KUKA KRL data list: ps_com_geo_c1.dat

&ACCESS RVO1
&REL 24
&COMMENT Solda GUN C1 Geometria
&PARAM DISKPATH = KRC:\R1\Program\SOLDA LTC
DEFDAT  ps_com_geo_c1
;FOLD EXTERNAL DECLARATIONS;%{PE}%MKUKATPBASIS,%CEXT,%VCOMMON,%P
;FOLD GRIPPERTECH EXT
EXT  H50 (INT  :IN,INT  :IN,INT  :IN,GRP_TYP  :IN )
;ENDFOLD (GRIPPERTECH EXT)
;FOLD SPOTTECH EXT
EXT  USERSPOT (S_COMMAND  :IN,SPOT_TYPE  :IN )
;ENDFOLD (SPOTTECH EXT)
;FOLD BASISTECH EXT;%{PE}%MKUKATPBASIS,%CEXT,%VEXT,%P
EXT  BAS (BAS_COMMAND  :IN,REAL  :IN )
DECL INT SUCCESS
;ENDFOLD (BASISTECH EXT)
;FOLD USER EXT;%{E}%MKUKATPUSER,%CEXT,%VEXT,%P
;Make your modifications here

;ENDFOLD (USER EXT)
;ENDFOLD (EXTERNAL DECLARATIONS)

;# ============ START PATH : swp_p13050r4_com_geo_c1 =============
DECL FDAT Fs_lx488={TOOL_NO 1,BASE_NO 1,IPO_FRAME #BASE,POINT2[] " "}
DECL PDAT PP_OLP5={VEL 100.0,ACC 100.0,APO_DIST 100.0,APO_MODE #CDIS}
DECL E6POS Xs_lx488={X -360.817993,Y 965.559021,Z 683.950989,A 93.2594986,B 64.8991013,C -75.3226013,S 2,T 10,E1 4060.29907,E2 0.0,E3 0.0,E4 0.0,E5 0.0,E6 0.0}
DECL FDAT Fswp_60_5140={TOOL_NO 1,BASE_NO 1,IPO_FRAME #BASE,POINT2[] " "}
DECL PDAT PP_OLP7={VEL 100.0,ACC 100.0,APO_DIST 0.0}
DECL SPOT_TYPE SS_OLP1={GUN 1,PAIR #FIRST,RETR #CLO,CLO_TM 0,PGNO1 1,PRESS1 1.0,PGNO2 0,PRESS2 0.0}
DECL E6POS Xswp_60_5140={X 136.687195,Y 902.795288,Z 579.572021,A 83.2147293,B 65.6525803,C -84.4438324,S 2,T 10,E1 4060.30103,E2 0.0,E3 0.0,E4 0.0,E5 0.0,E6 0.0}
DECL FDAT Fs_lx486={TOOL_NO 1,BASE_NO 1,IPO_FRAME #BASE,POINT2[] " "}
DECL PDAT PP_OLP9={VEL 100.0,ACC 100.0,APO_DIST 100.0,APO_MODE #CDIS}
DECL E6POS Xs_lx486={X -360.820007,Y 965.559998,Z 683.950989,A 93.2594986,B 64.8992004,C -75.3226013,S 2,T 10,E1 4060.29907,E2 0.0,E3 0.0,E4 0.0,E5 0.0,E6 0.0}
DECL PDAT PP_OLP10={VEL 100.0,ACC 100.0,APO_DIST 50.0,APO_MODE #CDIS}
DECL FDAT Fswp_60_5118={TOOL_NO 1,BASE_NO 1,IPO_FRAME #BASE,POINT2[] " "}
DECL PDAT PP_OLP12={VEL 100.0,ACC 100.0,APO_DIST 0.0}
DECL SPOT_TYPE SS_OLP2={GUN 1,PAIR #FIRST,RETR #CLO,CLO_TM 0,PGNO1 1,PRESS1 1.0,PGNO2 0,PRESS2 0.0}
DECL E6POS Xswp_60_5118={X 94.381012,Y 322.608704,Z 577.968018,A 0.639736116,B 88.9835663,C -175.218796,S 2,T 10,E1 4060.29199,E2 0.0,E3 0.0,E4 0.0,E5 0.0,E6 0.0}
DECL PDAT PP_OLP14={VEL 100.0,ACC 100.0,APO_DIST 100.0,APO_MODE #CDIS}
DECL PDAT PP_OLP16={VEL 100.0,ACC 100.0,APO_DIST 100.0,APO_MODE #CDIS}
DECL FDAT Fswp_60_5026={TOOL_NO 1,BASE_NO 1,IPO_FRAME #BASE,POINT2[] " "}
DECL PDAT PP_OLP18={VEL 100.0,ACC 100.0,APO_DIST 0.0}
DECL SPOT_TYPE SS_OLP3={GUN 1,PAIR #FIRST,RETR #CLO,CLO_TM 0,PGNO1 1,PRESS1 1.0,PGNO2 0,PRESS2 0.0}
DECL E6POS Xswp_60_5026={X 159.332901,Y 427.524109,Z 4.32035685,A 90.0029831,B -50.8949509,C -90.0011292,S 2,T 42,E1 4060.2771,E2 0.0,E3 0.0,E4 0.0,E5 0.0,E6 0.0}
DECL FDAT Fswp_60_5020={TOOL_NO 1,BASE_NO 1,IPO_FRAME #BASE,POINT2[] " "}
DECL PDAT PP_OLP19={VEL 100.0,ACC 100.0,APO_DIST 0.0}
DECL SPOT_TYPE SS_OLP4={GUN 1,PAIR #FIRST,RETR #CLO,CLO_TM 0,PGNO1 1,PRESS1 1.0,PGNO2 0,PRESS2 0.0}
DECL E6POS Xswp_60_5020={X 158.871796,Y 329.765594,Z 2.61356592,A 90.0077286,B -48.4540215,C -90.0015869,S 2,T 42,E1 4060.2981,E2 0.0,E3 0.0,E4 0.0,E5 0.0,E6 0.0}
DECL FDAT Fswp_60_5016={TOOL_NO 1,BASE_NO 1,IPO_FRAME #BASE,POINT2[] " "}
DECL PDAT PP_OLP20={VEL 100.0,ACC 100.0,APO_DIST 0.0}
DECL SPOT_TYPE SS_OLP5={GUN 1,PAIR #FIRST,RETR #CLO,CLO_TM 0,PGNO1 1,PRESS1 1.0,PGNO2 0,PRESS2 0.0}
DECL E6POS Xswp_60_5016={X 159.657196,Y 262.3927,Z 3.53638506,A 90.0078125,B -48.4543304,C -90.0026169,S 2,T 42,E1 4060.2959,E2 0.0,E3 0.0,E4 0.0,E5 0.0,E6 0.0}
DECL FDAT Fswp_60_5014={TOOL_NO 1,BASE_NO 1,IPO_FRAME #BASE,POINT2[] " "}
DECL PDAT PP_OLP21={VEL 100.0,ACC 100.0,APO_DIST 0.0}
DECL SPOT_TYPE SS_OLP6={GUN 1,PAIR #FIRST,RETR #CLO,CLO_TM 0,PGNO1 1,PRESS1 1.0,PGNO2 0,PRESS2 0.0}
DECL E6POS Xswp_60_5014={X 159.661102,Y 231.6185,Z 3.63049507,A 90.0080414,B -48.4544716,C -90.0028687,S 2,T 42,E1 4060.29712,E2 0.0,E3 0.0,E4 0.0,E5 0.0,E6 0.0}
DECL PDAT PP_OLP22={VEL 100.0,ACC 100.0,APO_DIST 100.0,APO_MODE #CDIS}
DECL FDAT Fs_lx470={TOOL_NO 1,BASE_NO 1,IPO_FRAME #BASE,POINT2[] " "}
DECL PDAT PP_OLP23={VEL 100.0,ACC 100.0,APO_DIST 100.0,APO_MODE #CDIS}
DECL E6POS Xs_lx470={X -243.503998,Y 293.677002,Z -34.257,A 90.0,B -44.5937996,C -90.0,S 2,T 10,E1 4060.29907,E2 0.0,E3 0.0,E4 0.0,E5 0.0,E6 0.0}
DECL PDAT PP_OLP24={VEL 100.0,ACC 100.0,APO_DIST 100.0,APO_MODE #CDIS}
DECL FDAT Flx507={TOOL_NO 1,BASE_NO 1,IPO_FRAME #BASE,POINT2[] " "}
DECL PDAT PP_OLP25={VEL 100.0,ACC 100.0,APO_DIST 100.0,APO_MODE #CDIS}
DECL E6POS Xlx507={X -11.6990004,Y 1057.32996,Z -233.384003,A 68.1399002,B -45.7775993,C -90.0,S 2,T 10,E1 4060.29907,E2 0.0,E3 0.0,E4 0.0,E5 0.0,E6 0.0}
DECL PDAT PP_OLP26={VEL 100.0,ACC 100.0,APO_DIST 100.0,APO_MODE #CDIS}
DECL FDAT Fswp_60_5042={TOOL_NO 1,BASE_NO 1,IPO_FRAME #BASE,POINT2[] " "}
DECL PDAT PP_OLP27={VEL 100.0,ACC 100.0,APO_DIST 0.0}
DECL SPOT_TYPE SS_OLP7={GUN 1,PAIR #FIRST,RETR #CLO,CLO_TM 0,PGNO1 1,PRESS1 1.0,PGNO2 0,PRESS2 0.0}
DECL E6POS Xswp_60_5042={X 176.981293,Y 1036.93799,Z -181.563095,A 68.1404114,B -45.7783699,C -90.0011597,S 2,T 10,E1 4060.30005,E2 0.0,E3 0.0,E4 0.0,E5 0.0,E6 0.0}
DECL FDAT Fswp_60_5040={TOOL_NO 1,BASE_NO 1,IPO_FRAME #BASE,POINT2[] " "}
DECL PDAT PP_OLP28={VEL 100.0,ACC 100.0,APO_DIST 0.0}
DECL SPOT_TYPE SS_OLP8={GUN 1,PAIR #FIRST,RETR #CLO,CLO_TM 0,PGNO1 1,PRESS1 1.0,PGNO2 0,PRESS2 0.0}
DECL E6POS Xswp_60_5040={X 172.178604,Y 1008.79102,Z -183.401794,A 176.628098,B -88.2014084,C 167.694305,S 2,T 10,E1 4060.30103,E2 0.0,E3 0.0,E4 0.0,E5 0.0,E6 0.0}
DECL FDAT Fswp_60_5038={TOOL_NO 1,BASE_NO 1,IPO_FRAME #BASE,POINT2[] " "}
DECL PDAT PP_OLP29={VEL 100.0,ACC 100.0,APO_DIST 0.0}
DECL SPOT_TYPE SS_OLP9={GUN 1,PAIR #FIRST,RETR #CLO,CLO_TM 0,PGNO1 1,PRESS1 1.0,PGNO2 0,PRESS2 0.0}
DECL E6POS Xswp_60_5038={X 164.622696,Y 982.143127,Z -183.500595,A -120.116699,B -89.1609726,C 109.444,S 2,T 10,E1 4060.29907,E2 0.0,E3 0.0,E4 0.0,E5 0.0,E6 0.0}
DECL FDAT Fswp_60_5036={TOOL_NO 1,BASE_NO 1,IPO_FRAME #BASE,POINT2[] " "}
DECL SPOT_TYPE SS_OLP10={GUN 1,PAIR #FIRST,RETR #CLO,CLO_TM 0,PGNO1 1,PRESS1 1.0,PGNO2 0,PRESS2 0.0}
DECL E6POS Xswp_60_5036={X 179.731094,Y 901.85553,Z -137.682495,A -105.0299,B -89.9987488,C 105.028702,S 2,T 42,E1 4060.29907,E2 0.0,E3 0.0,E4 0.0,E5 0.0,E6 0.0}
DECL FDAT Fswp_60_5028={TOOL_NO 1,BASE_NO 1,IPO_FRAME #BASE,POINT2[] " "}
DECL PDAT PP_OLP32={VEL 100.0,ACC 100.0,APO_DIST 0.0}
DECL SPOT_TYPE SS_OLP11={GUN 1,PAIR #FIRST,RETR #CLO,CLO_TM 0,PGNO1 1,PRESS1 1.0,PGNO2 0,PRESS2 0.0}
DECL E6POS Xswp_60_5028={X 182.583893,Y 794.820129,Z -47.8096008,A -163.747406,B -89.5717773,C 163.750702,S 2,T 42,E1 4060.29395,E2 0.0,E3 0.0,E4 0.0,E5 0.0,E6 0.0}
DECL FDAT Fs_lx464={TOOL_NO 1,BASE_NO 1,IPO_FRAME #BASE,POINT2[] " "}
DECL PDAT PP_OLP33={VEL 100.0,ACC 100.0,APO_DIST 100.0,APO_MODE #CDIS}
DECL E6POS Xs_lx464={X 178.498993,Y 805.025024,Z -118.82,A 0.0,B -90.0,C 0.0,S 2,T 42,E1 4060.29907,E2 0.0,E3 0.0,E4 0.0,E5 0.0,E6 0.0}
DECL PDAT PP_OLP34={VEL 100.0,ACC 100.0,APO_DIST 100.0,APO_MODE #CDIS}
DECL SPOT_TYPE SS_OLP12={GUN 1,PAIR #FIRST,RETR #CLO,CLO_TM 0,PGNO1 1,PRESS1 1.0,PGNO2 0,PRESS2 0.0}
DECL FDAT Fswp_60_5203={TOOL_NO 1,BASE_NO 1,IPO_FRAME #BASE,POINT2[] " "}
DECL SPOT_TYPE SS_OLP13={GUN 1,PAIR #FIRST,RETR #CLO,CLO_TM 0,PGNO1 1,PRESS1 1.0,PGNO2 0,PRESS2 0.0}
DECL E6POS Xswp_60_5203={X 156.1819,Y 485.568604,Z 388.023712,A 90.0274734,B -54.6427803,C -86.9009323,S 2,T 10,E1 4060.31592,E2 0.0,E3 0.0,E4 0.0,E5 0.0,E6 0.0}
DECL FDAT Fswp_60_5195={TOOL_NO 1,BASE_NO 1,IPO_FRAME #BASE,POINT2[] " "}
DECL SPOT_TYPE SS_OLP14={GUN 1,PAIR #FIRST,RETR #CLO,CLO_TM 0,PGNO1 1,PRESS1 1.0,PGNO2 0,PRESS2 0.0}
DECL E6POS Xswp_60_5195={X 161.142303,Y 202.515198,Z 386.019104,A -88.2071686,B -36.5904808,C 88.8797302,S 2,T 10,E1 4060.31396,E2 0.0,E3 0.0,E4 0.0,E5 0.0,E6 0.0}
DECL FDAT Fswp_60_5190={TOOL_NO 1,BASE_NO 1,IPO_FRAME #BASE,POINT2[] " "}
DECL SPOT_TYPE SS_OLP15={GUN 1,PAIR #FIRST,RETR #CLO,CLO_TM 0,PGNO1 1,PRESS1 1.0,PGNO2 0,PRESS2 0.0}
DECL E6POS Xswp_60_5190={X 161.480301,Y 148.9478,Z 280.717194,A -89.3926468,B -1.94816995,C 88.6738968,S 2,T 10,E1 4060.31494,E2 0.0,E3 0.0,E4 0.0,E5 0.0,E6 0.0}
DECL FDAT Fswp_60_5218={TOOL_NO 1,BASE_NO 1,IPO_FRAME #BASE,POINT2[] " "}
DECL SPOT_TYPE SS_OLP16={GUN 1,PAIR #FIRST,RETR #CLO,CLO_TM 0,PGNO1 1,PRESS1 1.0,PGNO2 0,PRESS2 0.0}
DECL E6POS Xswp_60_5218={X 164.738403,Y 122.212402,Z 106.1138,A -90.9965591,B 31.5576591,C 87.71698,S 2,T 10,E1 4060.31396,E2 0.0,E3 0.0,E4 0.0,E5 0.0,E6 0.0}
DECL PDAT PP_OLP52={VEL 100.0,ACC 100.0,APO_DIST 100.0,APO_MODE #CDIS}
DECL SPOT_TYPE SS_OLP17={GUN 1,PAIR #FIRST,RETR #CLO,CLO_TM 0,PGNO1 1,PRESS1 1.0,PGNO2 0,PRESS2 0.0}
DECL SPOT_TYPE SS_OLP18={GUN 1,PAIR #FIRST,RETR #CLO,CLO_TM 0,PGNO1 1,PRESS1 1.0,PGNO2 0,PRESS2 0.0}
DECL SPOT_TYPE SS_OLP19={GUN 1,PAIR #FIRST,RETR #CLO,CLO_TM 0,PGNO1 1,PRESS1 1.0,PGNO2 0,PRESS2 0.0}
DECL FDAT Fswp_60_5066={TOOL_NO 1,BASE_NO 1,IPO_FRAME #BASE,POINT2[] " "}
DECL SPOT_TYPE SS_OLP20={GUN 1,PAIR #FIRST,RETR #CLO,CLO_TM 0,PGNO1 1,PRESS1 1.0,PGNO2 0,PRESS2 0.0}
DECL E6POS Xswp_60_5066={X 151.353302,Y 626.425415,Z 250.5159,A -92.1195831,B 18.5633907,C 91.8053436,S 2,T 10,E1 4060.30591,E2 0.0,E3 0.0,E4 0.0,E5 0.0,E6 0.0}
DECL PDAT PP_OLP59={VEL 100.0,ACC 100.0,APO_DIST 20.0,APO_MODE #CDIS}
DECL PDAT PP_OLP60={VEL 100.0,ACC 100.0,APO_DIST 20.0,APO_MODE #CDIS}
DECL PDAT PP_OLP61={VEL 100.0,ACC 100.0,APO_DIST 20.0,APO_MODE #CDIS}
DECL FDAT Fswp_60_5076={TOOL_NO 1,BASE_NO 1,IPO_FRAME #BASE,POINT2[] " "}
DECL PDAT PP_OLP63={VEL 100.0,ACC 100.0,APO_DIST 0.0}
DECL SPOT_TYPE SS_OLP21={GUN 1,PAIR #FIRST,RETR #CLO,CLO_TM 0,PGNO1 1,PRESS1 1.0,PGNO2 0,PRESS2 0.0}
DECL E6POS Xswp_60_5076={X 154.796707,Y 782.258972,Z 101.740097,A 87.1909637,B 70.1359329,C -93.0589066,S 2,T 10,E1 4060.29199,E2 0.0,E3 0.0,E4 0.0,E5 0.0,E6 0.0}
DECL PDAT PP_OLP64={VEL 100.0,ACC 100.0,APO_DIST 100.0,APO_MODE #CDIS}
DECL SPOT_TYPE SS_OLP22={GUN 1,PAIR #FIRST,RETR #CLO,CLO_TM 0,PGNO1 1,PRESS1 1.0,PGNO2 0,PRESS2 0.0}
DECL PDAT PP_OLP69={VEL 100.0,ACC 100.0,APO_DIST 100.0,APO_MODE #CDIS}
DECL PDAT PP_OLP72={VEL 100.0,ACC 100.0,APO_DIST 100.0,APO_MODE #CDIS}
DECL FDAT Fswp_60_5626={TOOL_NO 1,BASE_NO 1,IPO_FRAME #BASE,POINT2[] " "}
DECL PDAT PP_OLP73={VEL 100.0,ACC 100.0,APO_DIST 0.0}
DECL SPOT_TYPE SS_OLP23={GUN 1,PAIR #FIRST,RETR #CLO,CLO_TM 0,PGNO1 1,PRESS1 1.0,PGNO2 0,PRESS2 0.0}
DECL E6POS Xswp_60_5626={X 634.33252,Y 1098.11096,Z 1372.00806,A -179.633102,B -69.9991837,C 90.5753021,S 2,T 2,E1 5254.49902,E2 0.0,E3 0.0,E4 0.0,E5 0.0,E6 0.0}
DECL FDAT Fswp_60_5640={TOOL_NO 1,BASE_NO 1,IPO_FRAME #BASE,POINT2[] " "}
DECL PDAT PP_OLP74={VEL 100.0,ACC 100.0,APO_DIST 0.0}
DECL SPOT_TYPE SS_OLP24={GUN 1,PAIR #FIRST,RETR #CLO,CLO_TM 0,PGNO1 1,PRESS1 1.0,PGNO2 0,PRESS2 0.0}
DECL E6POS Xswp_60_5640={X 731.3703,Y 1097.53699,Z 1377.57104,A 0.929155171,B -80.0200806,C -89.9900208,S 2,T 2,E1 5254.5,E2 0.0,E3 0.0,E4 0.0,E5 0.0,E6 0.0}
DECL PDAT PP_OLP75={VEL 100.0,ACC 100.0,APO_DIST 100.0,APO_MODE #CDIS}
DECL PDAT PP_OLP76={VEL 100.0,ACC 100.0,APO_DIST 100.0,APO_MODE #CDIS}
DECL PDAT PP_OLP77={VEL 100.0,ACC 100.0,APO_DIST 50.0,APO_MODE #CDIS}
DECL PDAT PP_OLP78={VEL 100.0,ACC 100.0,APO_DIST 50.0,APO_MODE #CDIS}
DECL FDAT Fswp_60_5060={TOOL_NO 1,BASE_NO 1,IPO_FRAME #BASE,POINT2[] " "}
DECL PDAT PP_OLP79={VEL 100.0,ACC 100.0,APO_DIST 0.0}
DECL SPOT_TYPE SS_OLP25={GUN 1,PAIR #FIRST,RETR #CLO,CLO_TM 0,PGNO1 1,PRESS1 1.0,PGNO2 0,PRESS2 0.0}
DECL E6POS Xswp_60_5060={X 440.014313,Y 1093.56006,Z -44.92976,A -177.803696,B 33.6436501,C 90.0005798,S 2,T 34,E1 5251.46289,E2 0.0,E3 0.0,E4 0.0,E5 0.0,E6 0.0}
DECL PDAT PP_OLP80={VEL 100.0,ACC 100.0,APO_DIST 50.0,APO_MODE #CDIS}
DECL PDAT PP_OLP81={VEL 100.0,ACC 100.0,APO_DIST 50.0,APO_MODE #CDIS}
DECL PDAT PP_OLP82={VEL 100.0,ACC 100.0,APO_DIST 100.0,APO_MODE #CDIS}
DECL FDAT Fswp_60_5056={TOOL_NO 1,BASE_NO 1,IPO_FRAME #BASE,POINT2[] " "}
DECL PDAT PP_OLP85={VEL 100.0,ACC 100.0,APO_DIST 0.0}
DECL SPOT_TYPE SS_OLP26={GUN 1,PAIR #FIRST,RETR #CLO,CLO_TM 0,PGNO1 1,PRESS1 1.0,PGNO2 0,PRESS2 0.0}
DECL E6POS Xswp_60_5056={X 372.068909,Y 1092.44397,Z -181.150497,A 178.998093,B -2.52557802,C 89.9496765,S 2,T 34,E1 5252.67188,E2 0.0,E3 0.0,E4 0.0,E5 0.0,E6 0.0}
DECL FDAT Fswp_60_5058={TOOL_NO 1,BASE_NO 1,IPO_FRAME #BASE,POINT2[] " "}
DECL PDAT PP_OLP86={VEL 100.0,ACC 100.0,APO_DIST 0.0}
DECL SPOT_TYPE SS_OLP27={GUN 1,PAIR #FIRST,RETR #CLO,CLO_TM 0,PGNO1 1,PRESS1 1.0,PGNO2 0,PRESS2 0.0}
DECL E6POS Xswp_60_5058={X 404.384796,Y 1091.41699,Z -160.593002,A 178.922501,B -10.25455,C 90.7412491,S 2,T 34,E1 5253.80078,E2 0.0,E3 0.0,E4 0.0,E5 0.0,E6 0.0}
DECL PDAT PP_OLP88={VEL 100.0,ACC 100.0,APO_DIST 100.0,APO_MODE #CDIS}
DECL PDAT PP_OLP89={VEL 100.0,ACC 100.0,APO_DIST 100.0,APO_MODE #CDIS}
DECL FDAT Fswp_60_5424={TOOL_NO 1,BASE_NO 1,IPO_FRAME #BASE,POINT2[] " "}
DECL PDAT PP_OLP91={VEL 100.0,ACC 100.0,APO_DIST 0.0}
DECL SPOT_TYPE SS_OLP28={GUN 1,PAIR #FIRST,RETR #CLO,CLO_TM 0,PGNO1 1,PRESS1 1.0,PGNO2 0,PRESS2 0.0}
DECL E6POS Xswp_60_5424={X 1302.37805,Y 1186.15405,Z -56.5237999,A -0.546349108,B -50.1205597,C -90.0004196,S 2,T 2,E1 5251.78613,E2 0.0,E3 0.0,E4 0.0,E5 0.0,E6 0.0}
DECL PDAT PP_OLP92={VEL 100.0,ACC 100.0,APO_DIST 100.0,APO_MODE #CDIS}
DECL PDAT PP_OLP93={VEL 100.0,ACC 100.0,APO_DIST 100.0,APO_MODE #CDIS}
DECL PDAT PP_OLP96={VEL 100.0,ACC 100.0,APO_DIST 100.0,APO_MODE #CDIS}
DECL PDAT PP_OLP97={VEL 100.0,ACC 100.0,APO_DIST 20.0,APO_MODE #CDIS}
DECL FDAT Fswp_60_5430={TOOL_NO 1,BASE_NO 1,IPO_FRAME #BASE,POINT2[] " "}
DECL PDAT PP_OLP100={VEL 100.0,ACC 100.0,APO_DIST 0.0}
DECL SPOT_TYPE SS_OLP29={GUN 1,PAIR #FIRST,RETR #CLO,CLO_TM 0,PGNO1 1,PRESS1 1.0,PGNO2 0,PRESS2 0.0}
DECL E6POS Xswp_60_5430={X 1286.38098,Y 1123.69702,Z 5.72508383,A -0.644820571,B 48.2571411,C -90.0793915,S 2,T 2,E1 6178.22119,E2 0.0,E3 0.0,E4 0.0,E5 0.0,E6 0.0}
DECL FDAT Fswp_60_5432={TOOL_NO 1,BASE_NO 1,IPO_FRAME #BASE,POINT2[] " "}
DECL PDAT PP_OLP101={VEL 100.0,ACC 100.0,APO_DIST 0.0}
DECL SPOT_TYPE SS_OLP30={GUN 1,PAIR #FIRST,RETR #CLO,CLO_TM 0,PGNO1 1,PRESS1 1.0,PGNO2 0,PRESS2 0.0}
DECL E6POS Xswp_60_5432={X 1304.38,Y 1123.71106,Z 21.1026192,A -0.644798875,B 48.25737,C -90.0797424,S 2,T 2,E1 6217.10498,E2 0.0,E3 0.0,E4 0.0,E5 0.0,E6 0.0}
DECL FDAT Fswp_60_5434={TOOL_NO 1,BASE_NO 1,IPO_FRAME #BASE,POINT2[] " "}
DECL PDAT PP_OLP102={VEL 100.0,ACC 100.0,APO_DIST 0.0}
DECL SPOT_TYPE SS_OLP31={GUN 1,PAIR #FIRST,RETR #CLO,CLO_TM 0,PGNO1 1,PRESS1 1.0,PGNO2 0,PRESS2 0.0}
DECL E6POS Xswp_60_5434={X 1288.31995,Y 1122.44202,Z 30.7160091,A -0.641988695,B 48.2577095,C -90.0761871,S 2,T 2,E1 6172.71387,E2 0.0,E3 0.0,E4 0.0,E5 0.0,E6 0.0}
DECL FDAT Fswp_60_5436={TOOL_NO 1,BASE_NO 1,IPO_FRAME #BASE,POINT2[] " "}
DECL PDAT PP_OLP105={VEL 100.0,ACC 100.0,APO_DIST 0.0}
DECL SPOT_TYPE SS_OLP32={GUN 1,PAIR #FIRST,RETR #CLO,CLO_TM 0,PGNO1 1,PRESS1 1.0,PGNO2 0,PRESS2 0.0}
DECL E6POS Xswp_60_5436={X 1304.93005,Y 1120.12903,Z 80.8903885,A -0.630691886,B 29.8777504,C -90.0939484,S 2,T 2,E1 6169.68115,E2 0.0,E3 0.0,E4 0.0,E5 0.0,E6 0.0}
DECL FDAT Fswp_60_5438={TOOL_NO 1,BASE_NO 1,IPO_FRAME #BASE,POINT2[] " "}
DECL PDAT PP_OLP107={VEL 100.0,ACC 100.0,APO_DIST 0.0}
DECL SPOT_TYPE SS_OLP33={GUN 1,PAIR #FIRST,RETR #CLO,CLO_TM 0,PGNO1 1,PRESS1 1.0,PGNO2 0,PRESS2 0.0}
DECL E6POS Xswp_60_5438={X 1335.14502,Y 1125.09802,Z 99.5109024,A -0.583152175,B 19.4271107,C -90.0527191,S 2,T 2,E1 5977.15283,E2 0.0,E3 0.0,E4 0.0,E5 0.0,E6 0.0}
DECL FDAT Fswp_60_5440={TOOL_NO 1,BASE_NO 1,IPO_FRAME #BASE,POINT2[] " "}
DECL PDAT PP_OLP108={VEL 100.0,ACC 100.0,APO_DIST 0.0}
DECL SPOT_TYPE SS_OLP34={GUN 1,PAIR #FIRST,RETR #CLO,CLO_TM 0,PGNO1 1,PRESS1 1.0,PGNO2 0,PRESS2 0.0}
DECL E6POS Xswp_60_5440={X 1334.10596,Y 1122.04004,Z 140.932205,A -0.565891325,B -2.25514102,C -90.0501328,S 2,T 2,E1 5826.48584,E2 0.0,E3 0.0,E4 0.0,E5 0.0,E6 0.0}
DECL PDAT PP_OLP109={VEL 100.0,ACC 100.0,APO_DIST 100.0,APO_MODE #CDIS}
DECL PDAT PP_OLP110={VEL 100.0,ACC 100.0,APO_DIST 100.0,APO_MODE #CDIS}
DECL PDAT PP_OLP111={VEL 100.0,ACC 100.0,APO_DIST 100.0,APO_MODE #CDIS}
DECL PDAT PP_OLP112={VEL 100.0,ACC 100.0,APO_DIST 100.0,APO_MODE #CDIS}
DECL PDAT PP_OLP113={VEL 100.0,ACC 100.0,APO_DIST 0.0,APO_MODE #CDIS}
DECL BASIS_SUGG_T LAST_BASIS={POINT1[] "P0                      ",POINT2[] "P0                      ",CP_PARAMS[] "CPDAT0                  ",PTP_PARAMS[] "PDAT0                   ",CONT[] "                        ",CP_VEL[] "2.0                     ",PTP_VEL[] " 100                    ",SYNC_PARAMS[] "SYNCDAT                 ",SPL_NAME[] "S0                      "}
DECL FDAT FXs_lx487={TOOL_NO 1,BASE_NO 1,IPO_FRAME #BASE,POINT2[] " ",TQ_STATE FALSE}
DECL E6POS XXS_LX487={X 142.0215,Y 865.563782,Z 629.299988,A 92.7790527,B 65.0505371,C -75.8403931,S 2,T 10,E1 4060.29395,E2 0.0,E3 0.0,E4 0.0,E5 0.0,E6 0.0}
DECL PDAT PPDAT2={VEL 100.0,ACC 100.0,APO_DIST 100.0,APO_MODE #CDIS}
DECL E6POS XXS_LX502={X 142.021301,Y 865.560791,Z 629.294983,A 92.7791138,B 65.0502167,C -75.8401871,S 2,T 10,E1 4060.29395,E2 0.0,E3 0.0,E4 0.0,E5 0.0,E6 0.0}
DECL FDAT FXs_lx502={TOOL_NO 1,BASE_NO 1,IPO_FRAME #BASE,POINT2[] " ",TQ_STATE FALSE}
DECL PDAT PPDAT6={VEL 100.0,ACC 100.0,APO_DIST 100.0,APO_MODE #CDIS}
DECL E6POS XXS_LX484={X -406.284088,Y 364.974487,Z 582.284119,A -59.6039505,B 89.6699677,C 128.917496,S 2,T 10,E1 4060.2981,E2 0.0,E3 0.0,E4 0.0,E5 0.0,E6 0.0}
DECL FDAT FXs_lx484={TOOL_NO 1,BASE_NO 1,IPO_FRAME #BASE,POINT2[] " ",TQ_STATE FALSE}
DECL E6POS XXS_LX504={X 102.534103,Y 321.186096,Z 604.033508,A 152.166595,B 89.932457,C -19.8392105,S 2,T 10,E1 4060.30005,E2 0.0,E3 0.0,E4 0.0,E5 0.0,E6 0.0}
DECL FDAT FXs_lx504={TOOL_NO 1,BASE_NO 1,IPO_FRAME #BASE,POINT2[] " ",TQ_STATE FALSE}
DECL PDAT PPDAT8={VEL 100.0,ACC 100.0,APO_DIST 50.0,APO_MODE #CDIS}
DECL E6POS XXS_LX506={X 101.603203,Y 324.702209,Z 606.954773,A -105.589798,B 89.533989,C 82.46315,S 2,T 10,E1 4060.29907,E2 0.0,E3 0.0,E4 0.0,E5 0.0,E6 0.0}
DECL FDAT FXs_lx506={TOOL_NO 1,BASE_NO 1,IPO_FRAME #BASE,POINT2[] " ",TQ_STATE FALSE}
DECL PDAT PPDAT10={VEL 100.0,ACC 100.0,APO_DIST 100.0,APO_MODE #CDIS}
DECL E6POS XXS_LX482={X -401.920288,Y 344.626587,Z 598.098022,A -123.613403,B 89.7013168,C 73.3319473,S 2,T 10,E1 4060.2981,E2 0.0,E3 0.0,E4 0.0,E5 0.0,E6 0.0}
DECL FDAT FXs_lx482={TOOL_NO 1,BASE_NO 1,IPO_FRAME #BASE,POINT2[] " ",TQ_STATE FALSE}
DECL E6POS XXS_LX510={X 164.903503,Y 407.34549,Z -24.669241,A 90.0030136,B -50.8949699,C -90.0012512,S 2,T 42,E1 4060.2771,E2 0.0,E3 0.0,E4 0.0,E5 0.0,E6 0.0}
DECL FDAT FXs_lx510={TOOL_NO 1,BASE_NO 1,IPO_FRAME #BASE,POINT2[] " ",TQ_STATE FALSE}
DECL PDAT PPDAT14={VEL 100.0,ACC 100.0,APO_DIST 100.0,APO_MODE #CDIS}
DECL E6POS XXS_LX469={X 176.571396,Y 282.161896,Z -22.7473507,A 89.9942474,B -44.593441,C -89.9960175,S 2,T 42,E1 4060.30103,E2 0.0,E3 0.0,E4 0.0,E5 0.0,E6 0.0}
DECL FDAT FXs_lx469={TOOL_NO 1,BASE_NO 1,IPO_FRAME #BASE,POINT2[] " ",TQ_STATE FALSE}
DECL E6POS XXS_LX468={X -247.606094,Y 804.985718,Z -118.853699,A 19.7734299,B -89.9986496,C -19.7741909,S 2,T 42,E1 4060.29907,E2 0.0,E3 0.0,E4 0.0,E5 0.0,E6 0.0}
DECL FDAT FXs_lx468={TOOL_NO 1,BASE_NO 1,IPO_FRAME #BASE,POINT2[] " ",TQ_STATE FALSE}
DECL E6POS XXS_LX512={X 180.2099,Y 1013.57098,Z -191.423492,A -25.3134308,B -87.7871933,C 9.87290573,S 2,T 10,E1 4060.29907,E2 0.0,E3 0.0,E4 0.0,E5 0.0,E6 0.0}
DECL FDAT FXs_lx512={TOOL_NO 1,BASE_NO 1,IPO_FRAME #BASE,POINT2[] " ",TQ_STATE FALSE}
DECL PDAT PPDAT16={VEL 100.0,ACC 100.0,APO_DIST 100.0,APO_MODE #CDIS}
DECL E6POS XXS_LX514={X 200.297501,Y 951.728088,Z -170.494797,A -120.180603,B -89.1640396,C 109.508102,S 2,T 10,E1 4060.2981,E2 0.0,E3 0.0,E4 0.0,E5 0.0,E6 0.0}
DECL FDAT FXs_lx514={TOOL_NO 1,BASE_NO 1,IPO_FRAME #BASE,POINT2[] " ",TQ_STATE FALSE}
DECL PDAT PPDAT18={VEL 100.0,ACC 100.0,APO_DIST 100.0,APO_MODE #CDIS}
DECL E6POS XXS_LX465={X -260.471985,Y 805.001709,Z -118.772697,A 138.775497,B -89.9979477,C -138.775497,S 2,T 42,E1 4060.31104,E2 0.0,E3 0.0,E4 0.0,E5 0.0,E6 0.0}
DECL FDAT FXs_lx465={TOOL_NO 1,BASE_NO 1,IPO_FRAME #BASE,POINT2[] " ",TQ_STATE FALSE}
DECL E6POS XXLX510={X 198.537292,Y 907.492188,Z 358.6026,A 89.3582687,B -28.1856194,C -88.5561295,S 2,T 10,E1 4060.30005,E2 0.0,E3 0.0,E4 0.0,E5 0.0,E6 0.0}
DECL FDAT FXlx510={TOOL_NO 1,BASE_NO 1,IPO_FRAME #BASE,POINT2[] " ",TQ_STATE FALSE}
DECL E6POS XXS_LX456={X -359.326691,Y 798.908997,Z 114.357002,A 87.1922531,B 70.1376114,C -93.0576477,S 2,T 10,E1 4060.30396,E2 0.0,E3 0.0,E4 0.0,E5 0.0,E6 0.0}
DECL FDAT FXs_lx456={TOOL_NO 1,BASE_NO 1,IPO_FRAME #BASE,POINT2[] " ",TQ_STATE FALSE}
DECL E6POS XXS_LX455={X -1161.73706,Y 2536.57007,Z -258.942688,A -75.5931015,B -3.65610003,C -1.19887197,S 2,T 2,E1 4060.30005,E2 0.0,E3 0.0,E4 0.0,E5 0.0,E6 0.0}
DECL FDAT FXs_lx455={TOOL_NO 1,BASE_NO 1,IPO_FRAME #BASE,POINT2[] " ",TQ_STATE FALSE}
DECL E6POS XXS_LX449={X 694.406311,Y 1082.60999,Z 1348.03699,A 1.31180894,B -80.1795273,C -90.3731537,S 2,T 2,E1 5254.49707,E2 0.0,E3 0.0,E4 0.0,E5 0.0,E6 0.0}
DECL FDAT FXs_lx449={TOOL_NO 1,BASE_NO 1,IPO_FRAME #BASE,POINT2[] " ",TQ_STATE FALSE}
DECL E6POS XXS_LX447={X 711.179504,Y 1091.54102,Z 1352.49304,A 0.941952884,B -85.4546738,C -90.002861,S 2,T 2,E1 5254.49902,E2 0.0,E3 0.0,E4 0.0,E5 0.0,E6 0.0}
DECL FDAT FXs_lx447={TOOL_NO 1,BASE_NO 1,IPO_FRAME #BASE,POINT2[] " ",TQ_STATE FALSE}
DECL E6POS XXS_LX448={X 697.610718,Y 1743.328,Z 1372.71704,A 0.930606484,B -81.3462601,C -89.9841232,S 2,T 2,E1 5254.5,E2 0.0,E3 0.0,E4 0.0,E5 0.0,E6 0.0}
DECL FDAT FXs_lx448={TOOL_NO 1,BASE_NO 1,IPO_FRAME #BASE,POINT2[] " ",TQ_STATE FALSE}
DECL E6POS XXS_LX446={X 371.822113,Y 1600.547,Z 7.65825987,A -177.905502,B 2.046278,C 91.1621094,S 2,T 34,E1 5251.48584,E2 0.0,E3 0.0,E4 0.0,E5 0.0,E6 0.0}
DECL FDAT FXs_lx446={TOOL_NO 1,BASE_NO 1,IPO_FRAME #BASE,POINT2[] " ",TQ_STATE FALSE}
DECL E6POS XXS_LX445={X 424.494812,Y 1084.04297,Z 14.3757401,A -177.9991,B 7.22483206,C 89.9997635,S 2,T 34,E1 5251.43408,E2 0.0,E3 0.0,E4 0.0,E5 0.0,E6 0.0}
DECL FDAT FXs_lx445={TOOL_NO 1,BASE_NO 1,IPO_FRAME #BASE,POINT2[] " ",TQ_STATE FALSE}
DECL E6POS XXS_LX442={X 424.496094,Y 1084.04297,Z 14.3774099,A -177.998993,B 7.22493505,C 89.9998398,S 2,T 34,E1 5251.43408,E2 0.0,E3 0.0,E4 0.0,E5 0.0,E6 0.0}
DECL FDAT FXs_lx442={TOOL_NO 1,BASE_NO 1,IPO_FRAME #BASE,POINT2[] " ",TQ_STATE FALSE}
DECL E6POS XXS_LX444={X 371.822113,Y 1600.547,Z 7.65825987,A -177.905502,B 2.046278,C 91.1621094,S 2,T 34,E1 5251.48584,E2 0.0,E3 0.0,E4 0.0,E5 0.0,E6 0.0}
DECL FDAT FXs_lx444={TOOL_NO 1,BASE_NO 1,IPO_FRAME #BASE,POINT2[] " ",TQ_STATE FALSE}
DECL E6POS XXS_LX520={X 449.010986,Y 1058.51904,Z -203.744797,A -179.592407,B -0.526983023,C 88.4325333,S 2,T 34,E1 5247.50293,E2 0.0,E3 0.0,E4 0.0,E5 0.0,E6 0.0}
DECL FDAT FXs_lx520={TOOL_NO 1,BASE_NO 1,IPO_FRAME #BASE,POINT2[] " ",TQ_STATE FALSE}
DECL PDAT PPDAT24={VEL 100.0,ACC 100.0,APO_DIST 100.0,APO_MODE #CDIS}
DECL E6POS XXS_LX521={X 401.931091,Y 1092.10706,Z -181.568497,A 179.003494,B -2.52484202,C 89.9398193,S 2,T 34,E1 5252.71582,E2 0.0,E3 0.0,E4 0.0,E5 0.0,E6 0.0}
DECL FDAT FXs_lx521={TOOL_NO 1,BASE_NO 1,IPO_FRAME #BASE,POINT2[] " ",TQ_STATE FALSE}
DECL PDAT PPDAT25={VEL 100.0,ACC 100.0,APO_DIST 100.0,APO_MODE #CDIS}
DECL E6POS XXS_LX522={X 448.946808,Y 1058.54504,Z -203.671799,A -179.594101,B -0.524964929,C 88.4331894,S 2,T 34,E1 5254.93994,E2 0.0,E3 0.0,E4 0.0,E5 0.0,E6 0.0}
DECL FDAT FXs_lx522={TOOL_NO 1,BASE_NO 1,IPO_FRAME #BASE,POINT2[] " ",TQ_STATE FALSE}
DECL PDAT PPDAT26={VEL 100.0,ACC 100.0,APO_DIST 100.0,APO_MODE #CDIS}
DECL E6POS XXS_LX439={X 1275.48706,Y 1356.73999,Z -29.0001392,A -10.9303904,B -49.6493797,C -82.047081,S 2,T 2,E1 5253.81494,E2 0.0,E3 0.0,E4 0.0,E5 0.0,E6 0.0}
DECL FDAT FXs_lx439={TOOL_NO 1,BASE_NO 1,IPO_FRAME #BASE,POINT2[] " ",TQ_STATE FALSE}
DECL E6POS XXS_LX524={X 1273.81299,Y 1177.25403,Z -109.4813,A -0.543687284,B -50.1182213,C -90.0044937,S 2,T 2,E1 5254.08496,E2 0.0,E3 0.0,E4 0.0,E5 0.0,E6 0.0}
DECL FDAT FXs_lx524={TOOL_NO 1,BASE_NO 1,IPO_FRAME #BASE,POINT2[] " ",TQ_STATE FALSE}
DECL PDAT PPDAT28={VEL 100.0,ACC 100.0,APO_DIST 20.0,APO_MODE #CDIS}
DECL E6POS XXS_LX434={X 1246.71497,Y 1183.89099,Z -102.509003,A -0.541095018,B -50.1177406,C -89.9982834,S 2,T 2,E1 5254.50391,E2 0.0,E3 0.0,E4 0.0,E5 0.0,E6 0.0}
DECL FDAT FXs_lx434={TOOL_NO 1,BASE_NO 1,IPO_FRAME #BASE,POINT2[] " ",TQ_STATE FALSE}
DECL E6POS XXS_LX525={X 1310.61304,Y 1545.06897,Z 103.151604,A -0.480830699,B -25.6063499,C -90.1753235,S 2,T 2,E1 5255.80176,E2 0.0,E3 0.0,E4 0.0,E5 0.0,E6 0.0}
DECL FDAT FXs_lx525={TOOL_NO 1,BASE_NO 1,IPO_FRAME #BASE,POINT2[] " ",TQ_STATE FALSE}
DECL PDAT PPDAT29={VEL 100.0,ACC 100.0,APO_DIST 100.0,APO_MODE #CDIS}
DECL E6POS XXS_LX526={X 1300.245,Y 1113.05396,Z 132.605804,A -0.57613349,B -13.6800003,C -89.9665985,S 2,T 2,E1 5571.7251,E2 0.0,E3 0.0,E4 0.0,E5 0.0,E6 0.0}
DECL FDAT FXs_lx526={TOOL_NO 1,BASE_NO 1,IPO_FRAME #BASE,POINT2[] " ",TQ_STATE FALSE}
DECL PDAT PPDAT30={VEL 100.0,ACC 100.0,APO_DIST 100.0,APO_MODE #CDIS}
DECL E6POS XXS_LX527={X 1292.80896,Y 1157.88098,Z 128.380295,A -0.5843454,B -17.4577408,C -89.9393997,S 2,T 2,E1 5253.43018,E2 0.0,E3 0.0,E4 0.0,E5 0.0,E6 0.0}
DECL FDAT FXs_lx527={TOOL_NO 1,BASE_NO 1,IPO_FRAME #BASE,POINT2[] " ",TQ_STATE FALSE}
DECL PDAT PPDAT31={VEL 100.0,ACC 100.0,APO_DIST 100.0,APO_MODE #CDIS}
DECL E6POS XXS_LX430={X 1291.24805,Y 1109.12805,Z 61.5505905,A -0.626630723,B 38.7113304,C -90.0650787,S 2,T 2,E1 6193.23291,E2 0.0,E3 0.0,E4 0.0,E5 0.0,E6 0.0}
DECL FDAT FXs_lx430={TOOL_NO 1,BASE_NO 1,IPO_FRAME #BASE,POINT2[] " ",TQ_STATE FALSE}
DECL E6POS XXS_LX431={X 1348.521,Y 1113.70105,Z 126.297096,A -0.588395178,B 1.75486195,C -90.0525818,S 2,T 2,E1 6075.11279,E2 0.0,E3 0.0,E4 0.0,E5 0.0,E6 0.0}
DECL FDAT FXs_lx431={TOOL_NO 1,BASE_NO 1,IPO_FRAME #BASE,POINT2[] " ",TQ_STATE FALSE}
DECL E6POS XXS_LX531={X 1273.10303,Y 1112.27405,Z 24.7617607,A -0.640370071,B 48.2600288,C -90.0756378,S 2,T 2,E1 6193.8999,E2 0.0,E3 0.0,E4 0.0,E5 0.0,E6 0.0}
DECL FDAT FXs_lx531={TOOL_NO 1,BASE_NO 1,IPO_FRAME #BASE,POINT2[] " ",TQ_STATE FALSE}
DECL PDAT PPDAT35={VEL 100.0,ACC 100.0,APO_DIST 20.0,APO_MODE #CDIS}
DECL E6POS XXS_LX532={X 1273.09595,Y 1106.79504,Z 52.060009,A -0.639810324,B 48.2610283,C -90.0751572,S 2,T 2,E1 6194.7832,E2 0.0,E3 0.0,E4 0.0,E5 0.0,E6 0.0}
DECL FDAT FXs_lx532={TOOL_NO 1,BASE_NO 1,IPO_FRAME #BASE,POINT2[] " ",TQ_STATE FALSE}
DECL PDAT PPDAT36={VEL 100.0,ACC 100.0,APO_DIST 20.0,APO_MODE #CDIS}
DECL E6POS XXS_LX421={X 1331.45801,Y 1113.62903,Z 140.508896,A -0.564055204,B -2.25771308,C -90.0505371,S 2,T 2,E1 5568.8999,E2 0.0,E3 0.0,E4 0.0,E5 0.0,E6 0.0}
DECL FDAT FXs_lx421={TOOL_NO 1,BASE_NO 1,IPO_FRAME #BASE,POINT2[] " ",TQ_STATE FALSE}
DECL E6POS XXS_LX422={X 1331.448,Y 1113.62598,Z 140.487,A -0.555783629,B -11.4802704,C -90.0506668,S 2,T 2,E1 5571.7002,E2 0.0,E3 0.0,E4 0.0,E5 0.0,E6 0.0}
DECL FDAT FXs_lx422={TOOL_NO 1,BASE_NO 1,IPO_FRAME #BASE,POINT2[] " ",TQ_STATE FALSE}
DECL E6POS XXS_LX534={X 1299.18005,Y 1113.90601,Z 155.308502,A -0.544914484,B -21.6417103,C -90.0528717,S 2,T 2,E1 5573.82813,E2 0.0,E3 0.0,E4 0.0,E5 0.0,E6 0.0}
DECL FDAT FXs_lx534={TOOL_NO 1,BASE_NO 1,IPO_FRAME #BASE,POINT2[] " ",TQ_STATE FALSE}
DECL PDAT PPDAT38={VEL 100.0,ACC 100.0,APO_DIST 100.0,APO_MODE #CDIS}
DECL E6POS XXS_LX423={X 1306.81396,Y 1263.76501,Z 115.999001,A -0.54406321,B -21.6427498,C -90.0545502,S 2,T 2,E1 5568.5918,E2 0.0,E3 0.0,E4 0.0,E5 0.0,E6 0.0}
DECL FDAT FXs_lx423={TOOL_NO 1,BASE_NO 1,IPO_FRAME #BASE,POINT2[] " ",TQ_STATE FALSE}
DECL E6POS XXS_LX424={X 1320.97205,Y 1519.14905,Z 108.012299,A 3.05467892,B -22.00144,C -89.1234894,S 2,T 2,E1 5572.271,E2 0.0,E3 0.0,E4 0.0,E5 0.0,E6 0.0}
DECL FDAT FXs_lx424={TOOL_NO 1,BASE_NO 1,IPO_FRAME #BASE,POINT2[] " ",TQ_STATE FALSE}
DECL E6POS XXS_LX535={X 1198.70996,Y 2189.93896,Z 25.40662,A -20.8274899,B -45.1372185,C -39.3026886,S 2,T 2,E1 5081.13379,E2 0.0,E3 0.0,E4 0.0,E5 0.0,E6 0.0}
DECL FDAT FXs_lx535={TOOL_NO 1,BASE_NO 1,IPO_FRAME #BASE,POINT2[] " ",TQ_STATE FALSE}
DECL PDAT PPDAT39={VEL 100.0,ACC 100.0,APO_DIST 100.0,APO_MODE #CDIS}
DECL E6POS XXS_LX537={X -459.137207,Y 2830.60693,Z -400.969299,A -93.8874512,B -1.00689602,C -1.81860495,S 2,T 2,E1 3742.04102,E2 0.0,E3 0.0,E4 0.0,E5 0.0,E6 0.0}
DECL FDAT FXs_lx537={TOOL_NO 1,BASE_NO 1,IPO_FRAME #BASE,POINT2[] " ",TQ_STATE FALSE}
DECL PDAT PPDAT41={VEL 100.0,ACC 100.0,APO_DIST 100.0,APO_MODE #CDIS}
DECL E6POS XXS_LX386={X -5394.59424,Y 2817.8999,Z -52.6045113,A -87.9566803,B 0.248233899,C 10.3403301,S 2,T 2,E1 -351.032715,E2 0.0,E3 0.0,E4 0.0,E5 0.0,E6 0.0}
DECL FDAT FXs_lx386={TOOL_NO 1,BASE_NO 1,IPO_FRAME #BASE,POINT2[] " ",TQ_STATE FALSE}
DECL SPOT_SUGG_T LAST_SPOT={GUN[] "1                       ",RETR_CMD[] "#CLO                    ",CHOISE[] "#FIRST                  ",CLO_TM[] "1                       ",PGNO1[] "25                      ",PRESS1[] "0                       ",PGNO2[] "1                       ",PRESS2[] "0                       ",SPOT_PARAMS[] "NORMAL                  "}
DECL PDAT PPDAT45={VEL 100.0,ACC 100.0,APO_DIST 100.0}
DECL E6POS XXS_LX546={X -1347.76294,Y 876.430298,Z -504.167694,A 136.986801,B 12.0716896,C -14.1013803,S 2,T 10,E1 4060.2981,E2 0.0,E3 0.0,E4 0.0,E5 0.0,E6 0.0}
DECL FDAT FXs_lx546={TOOL_NO 1,BASE_NO 1,IPO_FRAME #BASE,POINT2[] " ",TQ_STATE FALSE}
DECL PDAT PPDAT51={VEL 100.0,ACC 100.0,APO_DIST 100.0,APO_MODE #CDIS}
DECL E6POS XXS_LX548={X -1567.92603,Y 1474.04395,Z -380.613098,A -176.587601,B 10.73598,C -5.45803499,S 2,T 10,E1 4060.2981,E2 0.0,E3 0.0,E4 0.0,E5 0.0,E6 0.0}
DECL FDAT FXs_lx548={TOOL_NO 1,BASE_NO 1,IPO_FRAME #BASE,POINT2[] " ",TQ_STATE FALSE}
DECL PDAT PPDAT53={VEL 100.0,ACC 100.0,APO_DIST 100.0}
DECL E6POS XXS_LX463={X -285.360809,Y 775.312988,Z 375.377014,A -91.1736984,B -86.1419373,C 91.3704376,S 2,T 42,E1 4059.50293,E2 0.0,E3 0.0,E4 0.0,E5 0.0,E6 0.0}
DECL FDAT FXs_lx463={TOOL_NO 1,BASE_NO 1,IPO_FRAME #BASE,POINT2[] " ",TQ_STATE FALSE}
DECL E6POS XXS_LX552={X -7591.26416,Y 3233.35889,Z -215.513107,A -30.6375008,B 9.25732231,C -0.711479485,S 2,T 11,E1 -353.282715,E2 0.0,E3 0.0,E4 0.0,E5 0.0,E6 0.0}
DECL FDAT FXs_lx552={TOOL_NO 1,BASE_NO 1,IPO_FRAME #BASE,POINT2[] " ",TQ_STATE FALSE}
DECL PDAT PPDAT57={VEL 100.0,ACC 100.0,APO_DIST 100.0,APO_MODE #CDIS}
DECL PDAT PP_OLP116={VEL 100.0,ACC 100.0,APO_DIST 100.0,APO_MODE #CDIS}
DECL E6POS Xc_lx33={X -5797.43311,Y 2784.89893,Z -341.750305,A -179.385498,B 9.2559042,C -0.711720884,S 2,T 10,E1 -353.282196,E2 0.0,E3 0.0,E4 0.0,E5 0.0,E6 0.0}
DECL FDAT Fc_lx33={TOOL_NO 1,BASE_NO 2,IPO_FRAME #BASE,POINT2[] " ",TQ_STATE FALSE}
DECL E6POS XP2={X -1008.41998,Y -3878.53809,Z 2280.71802,A 15.8486004,B 69.8013687,C 116.1772,S 2,T 10,E1 3309.09106,E2 0.0,E3 0.0,E4 0.0,E5 0.0,E6 0.0}
DECL FDAT FP2={TOOL_NO 8,BASE_NO 0,IPO_FRAME #BASE,POINT2[] " ",TQ_STATE FALSE}
DECL PDAT PPDAT58={VEL 100.0,ACC 100.0,APO_DIST 100.0}
DECL E6POS XP3={X -2899.04102,Y 3376.81909,Z 87.3140106,A -134.810806,B 53.134861,C -12.8320503,S 2,T 10,E1 2156.50293,E2 0.0,E3 0.0,E4 0.0,E5 0.0,E6 0.0}
DECL FDAT FP3={TOOL_NO 1,BASE_NO 2,IPO_FRAME #BASE,POINT2[] " ",TQ_STATE FALSE}
DECL PDAT PPDAT59={VEL 100.0,ACC 100.0,APO_DIST 100.0,APO_MODE #CDIS}
DECL E6POS XXS_LX472={X -406.190887,Y 292.545807,Z -34.1930313,A 73.3883972,B -43.3940392,C -82.1220627,S 2,T 10,E1 4060.30005,E2 0.0,E3 0.0,E4 0.0,E5 0.0,E6 0.0}
DECL FDAT FXs_lx472={TOOL_NO 1,BASE_NO 1,IPO_FRAME #BASE,POINT2[] " ",TQ_STATE FALSE}
DECL E6POS XXS_LX443={X 490.55899,Y 1425.50195,Z -219.291702,A -179.175095,B -0.318304598,C 84.957428,S 2,T 34,E1 5250.30322,E2 0.0,E3 0.0,E4 0.0,E5 0.0,E6 0.0}
DECL FDAT FXs_lx443={TOOL_NO 1,BASE_NO 1,IPO_FRAME #BASE,POINT2[] " ",TQ_STATE FALSE}
DECL E6POS XXS_LX437={X 735.744385,Y 1314.55798,Z -205.183502,A -177.910797,B -6.01889086,C 78.0020905,S 2,T 34,E1 5254.11084,E2 0.0,E3 0.0,E4 0.0,E5 0.0,E6 0.0}
DECL FDAT FXs_lx437={TOOL_NO 1,BASE_NO 1,IPO_FRAME #BASE,POINT2[] " ",TQ_STATE FALSE}
DECL E6POS XXS_LX435={X 1247.71399,Y 1296.47705,Z -102.5009,A -0.543420196,B -50.1155205,C -90.0,S 2,T 2,E1 5252.6582,E2 0.0,E3 0.0,E4 0.0,E5 0.0,E6 0.0}
DECL FDAT FXs_lx435={TOOL_NO 1,BASE_NO 1,IPO_FRAME #BASE,POINT2[] " ",TQ_STATE FALSE}
DECL E6POS XXS_LX467={X 171.180801,Y 983.950684,Z -233.371597,A 68.1400681,B -45.7760887,C -90.0009766,S 2,T 10,E1 4060.30103,E2 0.0,E3 0.0,E4 0.0,E5 0.0,E6 0.0}
DECL FDAT FXs_lx467={TOOL_NO 1,BASE_NO 1,IPO_FRAME #BASE,POINT2[] " ",TQ_STATE FALSE}
DECL E6POS XXLX511={X 202.229294,Y 896.270508,Z 253.845901,A 90.3564911,B 13.9303102,C -88.6880264,S 2,T 10,E1 4060.302,E2 0.0,E3 0.0,E4 0.0,E5 0.0,E6 0.0}
DECL FDAT FXlx511={TOOL_NO 1,BASE_NO 1,IPO_FRAME #BASE,POINT2[] " ",TQ_STATE FALSE}
DECL E6POS XXLX509={X 162.742096,Y 891.286621,Z 202.198807,A 89.3670578,B 33.9861488,C -91.2537766,S 2,T 10,E1 4060.302,E2 0.0,E3 0.0,E4 0.0,E5 0.0,E6 0.0}
DECL FDAT FXlx509={TOOL_NO 1,BASE_NO 1,IPO_FRAME #BASE,POINT2[] " ",TQ_STATE FALSE}
DECL PDAT PP_OLP118={VEL 100.0,ACC 100.0,APO_DIST 100.0,APO_MODE #CDIS}
DECL E6POS XXs_lx464={X 166.837997,Y 775.260925,Z 368.354614,A -91.1741104,B -86.1427383,C 91.370903,S 2,T 42,E1 4058.85107,E2 0.0,E3 0.0,E4 0.0,E5 0.0,E6 0.0}
DECL FDAT FXs_lx464={TOOL_NO 1,BASE_NO 1,IPO_FRAME #BASE,POINT2[] " ",TQ_STATE FALSE}
DECL PDAT PP_OLP119={VEL 100.0,ACC 100.0,APO_DIST 0.0}
DECL E6POS Xswp_60_5097={X 155.421204,Y 677.644409,Z 419.4534,A -89.9986191,B -76.7324066,C 89.9989395,S 2,T 42,E1 4060.29907,E2 0.0,E3 0.0,E4 0.0,E5 0.0,E6 0.0}
DECL FDAT Fswp_60_5097={TOOL_NO 1,BASE_NO 1,IPO_FRAME #BASE,POINT2[] " "}
DECL PDAT PP_OLP120={VEL 100.0,ACC 100.0,APO_DIST 0.0}
DECL E6POS Xswp_60_5099={X 155.171906,Y 756.641907,Z 420.422699,A 24.4609909,B -89.997139,C -24.46138,S 2,T 42,E1 4060.29907,E2 0.0,E3 0.0,E4 0.0,E5 0.0,E6 0.0}
DECL FDAT Fswp_60_5099={TOOL_NO 1,BASE_NO 1,IPO_FRAME #BASE,POINT2[] " "}
DECL PDAT PP_OLP121={VEL 100.0,ACC 100.0,APO_DIST 0.0}
DECL E6POS Xswp_60_5101={X 155.733994,Y 840.013794,Z 421.443298,A 24.8737907,B -89.9972229,C -24.8741093,S 2,T 42,E1 4060.29907,E2 0.0,E3 0.0,E4 0.0,E5 0.0,E6 0.0}
DECL FDAT Fswp_60_5101={TOOL_NO 1,BASE_NO 1,IPO_FRAME #BASE,POINT2[] " "}
DECL PDAT PP_OLP122={VEL 100.0,ACC 100.0,APO_DIST 0.0}
DECL E6POS Xswp_60_5085={X 156.082306,Y 894.531006,Z 254.542404,A 89.7875671,B 15.1001301,C -91.0752563,S 2,T 10,E1 4060.30103,E2 0.0,E3 0.0,E4 0.0,E5 0.0,E6 0.0}
DECL FDAT Fswp_60_5085={TOOL_NO 1,BASE_NO 1,IPO_FRAME #BASE,POINT2[] " "}
DECL E6POS XP8={X -291.032288,Y 1013.00403,Z -302.712006,A -102.734497,B 68.9540329,C 77.207077,S 2,T 10,E1 4060.31104,E2 0.0,E3 0.0,E4 0.0,E5 0.0,E6 0.0}
DECL FDAT FP8={TOOL_NO 1,BASE_NO 1,IPO_FRAME #BASE,POINT2[] " ",TQ_STATE FALSE}
DECL PDAT PPDAT65={VEL 100.0,ACC 100.0,APO_DIST 100.0,APO_MODE #CDIS}
DECL E6POS XP9={X -205.798492,Y 207.417007,Z 211.056396,A -93.6165237,B 13.9594002,C 90.2877808,S 2,T 10,E1 4060.31104,E2 0.0,E3 0.0,E4 0.0,E5 0.0,E6 0.0}
DECL FDAT FP9={TOOL_NO 1,BASE_NO 1,IPO_FRAME #BASE,POINT2[] " ",TQ_STATE FALSE}
DECL PDAT PPDAT66={VEL 100.0,ACC 100.0,APO_DIST 100.0,APO_MODE #CDIS}
DECL E6POS XP10={X 190.3022,Y 135.982407,Z 204.456207,A -96.1434937,B 14.1406603,C 89.6691132,S 2,T 10,E1 4060.31201,E2 0.0,E3 0.0,E4 0.0,E5 0.0,E6 0.0}
DECL FDAT FP10={TOOL_NO 1,BASE_NO 1,IPO_FRAME #BASE,POINT2[] " ",TQ_STATE FALSE}
DECL PDAT PPDAT67={VEL 100.0,ACC 100.0,APO_DIST 100.0,APO_MODE #CDIS}
DECL PDAT PPDAT68={VEL 100.0,ACC 100.0,APO_DIST 100.0}
DECL E6POS XP13={X 169.981796,Y 176.841797,Z 220.672104,A -89.7854614,B 11.5515804,C 87.9993362,S 2,T 10,E1 4060.31494,E2 0.0,E3 0.0,E4 0.0,E5 0.0,E6 0.0}
DECL FDAT FP13={TOOL_NO 1,BASE_NO 1,IPO_FRAME #BASE,POINT2[] " ",TQ_STATE FALSE}
DECL PDAT PPDAT70={VEL 100.0,ACC 100.0,APO_DIST 100.0,APO_MODE #CDIS}
DECL PDAT PPDAT71={VEL 100.0,ACC 100.0,APO_DIST 100.0}
DECL PDAT PPDAT72={VEL 100.0,ACC 100.0,APO_DIST 100.0,APO_MODE #CDIS}
DECL E6POS Xpt1={X 161.814499,Y 201.080795,Z 274.221313,A -88.7676163,B -26.3682098,C 88.4874115,S 2,T 10,E1 4060.31494,E2 0.0,E3 0.0,E4 0.0,E5 0.0,E6 0.0}
DECL FDAT Fpt1={TOOL_NO 1,BASE_NO 1,IPO_FRAME #BASE,POINT2[] " ",TQ_STATE FALSE}
DECL PDAT PPDAT73={VEL 100.0,ACC 100.0,APO_DIST 100.0}
DECL E6POS XPT2={X 159.854294,Y 242.701508,Z 357.2724,A -87.5249329,B -56.4212418,C 88.3794632,S 2,T 10,E1 4060.31592,E2 0.0,E3 0.0,E4 0.0,E5 0.0,E6 0.0}
DECL FDAT Fpt2={TOOL_NO 1,BASE_NO 1,IPO_FRAME #BASE,POINT2[] " ",TQ_STATE FALSE}
DECL PDAT PPDAT74={VEL 100.0,ACC 100.0,APO_DIST 100.0,APO_MODE #CDIS}
DECL E6POS XPT3={X 169.334305,Y 358.47821,Z 399.365112,A 87.187088,B -69.8794937,C -84.8208008,S 2,T 10,E1 4060.31592,E2 0.0,E3 0.0,E4 0.0,E5 0.0,E6 0.0}
DECL FDAT Fpt3={TOOL_NO 1,BASE_NO 1,IPO_FRAME #BASE,POINT2[] " ",TQ_STATE FALSE}
DECL PDAT PPDAT75={VEL 100.0,ACC 100.0,APO_DIST 100.0,APO_MODE #CDIS}
DECL PDAT PPDAT76={VEL 100.0,ACC 100.0,APO_DIST 100.0}
DECL E6POS XPT4={X 163.896896,Y 440.960114,Z 374.004089,A 88.4197922,B -54.7953987,C -86.9808578,S 2,T 10,E1 4060.31299,E2 0.0,E3 0.0,E4 0.0,E5 0.0,E6 0.0}
DECL FDAT Fpt4={TOOL_NO 1,BASE_NO 1,IPO_FRAME #BASE,POINT2[] " ",TQ_STATE FALSE}
DECL PDAT PPDAT77={VEL 100.0,ACC 100.0,APO_DIST 100.0}
DECL E6POS XPT5={X -312.486206,Y 433.580505,Z 388.477386,A 88.4197922,B -54.7953987,C -86.9808578,S 2,T 10,E1 4060.31299,E2 0.0,E3 0.0,E4 0.0,E5 0.0,E6 0.0}
DECL FDAT Fpt5={TOOL_NO 1,BASE_NO 1,IPO_FRAME #BASE,POINT2[] " ",TQ_STATE FALSE}
DECL PDAT PPDAT78={VEL 100.0,ACC 100.0,APO_DIST 100.0,APO_MODE #CDIS}
DECL E6POS XPT6={X -312.831299,Y 431.701508,Z 162.645004,A 96.246109,B 71.9801483,C -84.3668823,S 2,T 10,E1 4060.31299,E2 0.0,E3 0.0,E4 0.0,E5 0.0,E6 0.0}
DECL FDAT Fpt6={TOOL_NO 1,BASE_NO 1,IPO_FRAME #BASE,POINT2[] " ",TQ_STATE FALSE}
DECL PDAT PPDAT79={VEL 100.0,ACC 100.0,APO_DIST 100.0,APO_MODE #CDIS}
DECL E6POS XPT7={X 154.929993,Y 439.048096,Z 148.423401,A 93.5119171,B 56.3998604,C -86.8548965,S 2,T 10,E1 4060.30005,E2 0.0,E3 0.0,E4 0.0,E5 0.0,E6 0.0}
DECL FDAT Fpt7={TOOL_NO 1,BASE_NO 1,IPO_FRAME #BASE,POINT2[] " ",TQ_STATE FALSE}
DECL PDAT PPDAT80={VEL 100.0,ACC 100.0,APO_DIST 100.0,APO_MODE #CDIS}
DECL E6POS XSWP_60_5209={X 156.664795,Y 490.26001,Z 142.292603,A 93.5122604,B 56.3994598,C -86.8546371,S 2,T 10,E1 4060.30005,E2 0.0,E3 0.0,E4 0.0,E5 0.0,E6 0.0}
DECL FDAT Fswp_60_5209={TOOL_NO 1,BASE_NO 1,IPO_FRAME #BASE,POINT2[] " ",TQ_STATE FALSE}
DECL PDAT PPDAT81={VEL 100.0,ACC 100.0,APO_DIST 100.0}
DECL PDAT PPDAT82={VEL 100.0,ACC 100.0,APO_DIST 100.0}
DECL E6POS Xpt8={X 154.929993,Y 439.048096,Z 148.423401,A 93.5119171,B 56.3998604,C -86.8548965,S 2,T 10,E1 4060.30005,E2 0.0,E3 0.0,E4 0.0,E5 0.0,E6 0.0}
DECL FDAT Fpt8={TOOL_NO 1,BASE_NO 1,IPO_FRAME #BASE,POINT2[] " ",TQ_STATE FALSE}
DECL E6POS XPT9={X -312.831299,Y 431.701508,Z 162.645004,A 96.246109,B 71.9801483,C -84.3668823,S 2,T 10,E1 4060.31299,E2 0.0,E3 0.0,E4 0.0,E5 0.0,E6 0.0}
DECL FDAT Fpt9={TOOL_NO 1,BASE_NO 1,IPO_FRAME #BASE,POINT2[] " ",TQ_STATE FALSE}
DECL PDAT PPDAT83={VEL 100.0,ACC 100.0,APO_DIST 100.0}
DECL E6POS XPT11={X 160.858307,Y 725.869202,Z 118.343903,A -89.463562,B 67.0390701,C 92.8514862,S 2,T 10,E1 4060.30396,E2 0.0,E3 0.0,E4 0.0,E5 0.0,E6 0.0}
DECL FDAT Fpt11={TOOL_NO 1,BASE_NO 1,IPO_FRAME #BASE,POINT2[] " ",TQ_STATE FALSE}
DECL PDAT PPDAT85={VEL 100.0,ACC 100.0,APO_DIST 100.0,APO_MODE #CDIS}
DECL E6POS XPT12={X 161.1828,Y 693.768921,Z 161.033401,A -90.1003571,B 49.8515396,C 94.0767822,S 2,T 10,E1 4060.30396,E2 0.0,E3 0.0,E4 0.0,E5 0.0,E6 0.0}
DECL FDAT Fpt12={TOOL_NO 1,BASE_NO 1,IPO_FRAME #BASE,POINT2[] " ",TQ_STATE FALSE}
DECL PDAT PPDAT86={VEL 100.0,ACC 100.0,APO_DIST 100.0,APO_MODE #CDIS}
DECL E6POS XPT13={X 175.753799,Y 675.288574,Z 178.158401,A -90.3979263,B 47.0033798,C 94.2010193,S 2,T 10,E1 4060.30493,E2 0.0,E3 0.0,E4 0.0,E5 0.0,E6 0.0}
DECL FDAT Fpt13={TOOL_NO 1,BASE_NO 1,IPO_FRAME #BASE,POINT2[] " ",TQ_STATE FALSE}
DECL PDAT PPDAT87={VEL 100.0,ACC 100.0,APO_DIST 100.0,APO_MODE #CDIS}
DECL E6POS XPT14={X 179.009003,Y 617.818115,Z 251.7612,A -92.1164398,B 18.5910301,C 93.9508972,S 2,T 10,E1 4060.30493,E2 0.0,E3 0.0,E4 0.0,E5 0.0,E6 0.0}
DECL FDAT Fpt14={TOOL_NO 1,BASE_NO 1,IPO_FRAME #BASE,POINT2[] " ",TQ_STATE FALSE}
DECL PDAT PPDAT88={VEL 100.0,ACC 100.0,APO_DIST 100.0,APO_MODE #CDIS}
DECL PDAT PPDAT89={VEL 100.0,ACC 100.0,APO_DIST 100.0}
DECL E6POS XPT15={X 179.009003,Y 617.818115,Z 251.7612,A -92.1164398,B 18.5910301,C 93.9508972,S 2,T 10,E1 4060.30493,E2 0.0,E3 0.0,E4 0.0,E5 0.0,E6 0.0}
DECL FDAT Fpt15={TOOL_NO 1,BASE_NO 1,IPO_FRAME #BASE,POINT2[] " ",TQ_STATE FALSE}
DECL PDAT PPDAT90={VEL 100.0,ACC 100.0,APO_DIST 100.0}
DECL E6POS XPT16={X 175.753799,Y 675.288574,Z 178.158401,A -90.3979263,B 47.0033798,C 94.2010193,S 2,T 10,E1 4060.30493,E2 0.0,E3 0.0,E4 0.0,E5 0.0,E6 0.0}
DECL FDAT Fpt16={TOOL_NO 1,BASE_NO 1,IPO_FRAME #BASE,POINT2[] " ",TQ_STATE FALSE}
DECL PDAT PPDAT91={VEL 100.0,ACC 100.0,APO_DIST 100.0,APO_MODE #CDIS}
DECL E6POS XPT18={X 161.1828,Y 693.768921,Z 161.033401,A -90.1003571,B 49.8515396,C 94.0767822,S 2,T 10,E1 4060.30396,E2 0.0,E3 0.0,E4 0.0,E5 0.0,E6 0.0}
DECL FDAT Fpt18={TOOL_NO 1,BASE_NO 1,IPO_FRAME #BASE,POINT2[] " ",TQ_STATE FALSE}
DECL PDAT PPDAT93={VEL 100.0,ACC 100.0,APO_DIST 100.0,APO_MODE #CDIS}
DECL E6POS XPT19={X 160.822693,Y 729.790894,Z 127.590401,A -89.4637833,B 67.0392914,C 92.8511581,S 2,T 10,E1 4060.30396,E2 0.0,E3 0.0,E4 0.0,E5 0.0,E6 0.0}
DECL FDAT Fpt19={TOOL_NO 1,BASE_NO 1,IPO_FRAME #BASE,POINT2[] " ",TQ_STATE FALSE}
DECL PDAT PPDAT94={VEL 100.0,ACC 100.0,APO_DIST 100.0,APO_MODE #CDIS}
DECL E6POS XPT20={X 217.4048,Y 2369.823,Z -30.3654709,A -73.5321121,B -28.8238201,C -1.98111796,S 2,T 2,E1 4846.66211,E2 0.0,E3 0.0,E4 0.0,E5 0.0,E6 0.0}
DECL FDAT Fpt20={TOOL_NO 1,BASE_NO 1,IPO_FRAME #BASE,POINT2[] " ",TQ_STATE FALSE}
DECL PDAT PPDAT95={VEL 100.0,ACC 100.0,APO_DIST 100.0,APO_MODE #CDIS}
DECL E6POS XP14={X 673.541199,Y 1727.53601,Z 1378.01599,A 0.981028795,B -89.2553635,C -78.1354065,S 2,T 2,E1 5254.5,E2 0.0,E3 0.0,E4 0.0,E5 0.0,E6 0.0}
DECL FDAT FP14={TOOL_NO 1,BASE_NO 1,IPO_FRAME #BASE,POINT2[] " ",TQ_STATE FALSE}
DECL PDAT PPDAT96={VEL 100.0,ACC 100.0,APO_DIST 100.0,APO_MODE #CDIS}
DECL E6POS XP15={X 373.471985,Y 1712.46106,Z 714.465271,A 159.352203,B -72.0383682,C 115.424301,S 2,T 2,E1 5255.12988,E2 0.0,E3 0.0,E4 0.0,E5 0.0,E6 0.0}
DECL FDAT FP15={TOOL_NO 1,BASE_NO 1,IPO_FRAME #BASE,POINT2[] " ",TQ_STATE FALSE}
DECL PDAT PPDAT97={VEL 100.0,ACC 100.0,APO_DIST 100.0,APO_MODE #CDIS}
ENDDAT
